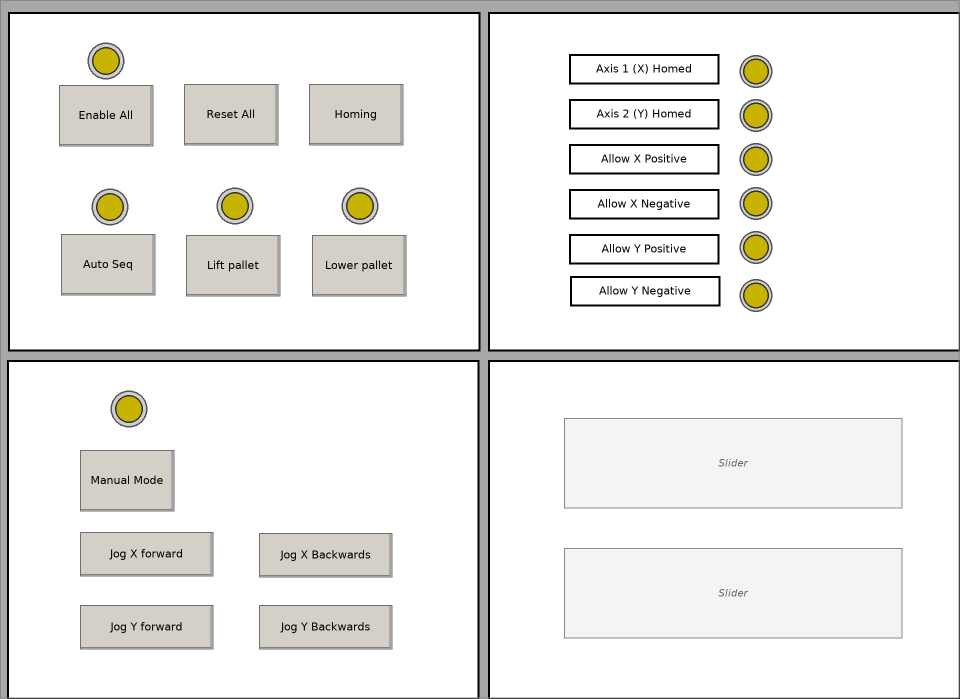
VISUALIZATION Visualization  // 960x699
    Rectangle (8,12 472x339)
    Rectangle (7,360 472x339)
    Rectangle (488,360 472x339)
    Rectangle (488,12 472x339)
    Button (59,85 94x61), "Enable All", colour toggle: GVL_Motion.bEnableAll, pressed state: GVL_Motion.bEnableAll
        OnMouseClick: toggle GVL_Motion.bEnableAll
    Button (184,84 94x61), "Reset All", colour toggle: GVL_Motion.bResetAll
        tap GVL_Motion.bResetAll
    Button (80,450 94x61), "Manual Mode", pressed state: GVL_Motion.bManualModeActive
        OnMouseClick: toggle GVL_Motion.bManualModeActive
    Button (61,234 94x61), "Auto Seq", pressed state: GVL_Motion.bStartAutoseq
        OnMouseClick: execute { GVL_Motion.bStartAutoseq := TRUE; }
    Button (309,84 94x61), "Homing", colour toggle: GVL_Motion.bStartHoming, pressed state: GVL_Motion.bStartHoming
        OnMouseClick: toggle GVL_Motion.bStartHoming
    Lamp1 (85,40 42x42), variable: GVL_Motion.bEnableAll, style: Lamp-Lamp1-Yellow
    Lamp1 (108,388 42x42), variable: GVL_Motion.bManualModeActive, style: Lamp-Lamp1-Yellow
    Button (80,532 133x44), "Jog X forward", pressed state: GVL_Motion.bJogForwardX
        OnMouseDown: toggle GVL_Motion.bJogForwardX
        OnMouseUp: toggle GVL_Motion.bJogForwardX
    Button (259,533 133x44), "Jog X Backwards", pressed state: GVL_Motion.bJogBackwardsX
        OnMouseDown: toggle GVL_Motion.bJogBackwardsX
        OnMouseUp: toggle GVL_Motion.bJogBackwardsX
    Button (80,605 133x44), "Jog Y forward", pressed state: GVL_Motion.bJogForwardY
        OnMouseDown: toggle GVL_Motion.bJogForwardY
        OnMouseUp: toggle GVL_Motion.bJogForwardY
    Button (259,605 133x44), "Jog Y Backwards", pressed state: GVL_Motion.bJogBackwardsY
        OnMouseDown: toggle GVL_Motion.bJogBackwardsY
        OnMouseUp: toggle GVL_Motion.bJogBackwardsY
    Slider (564,418 338x90), variable: GVL_Motion.fVelocityX, scale 0..30
    Slider (564,548 338x90), variable: GVL_Motion.fVelocityY, scale 0..30
    Lamp1 (737,52 38x39), variable: GVL_Motion.bXHomed, style: Lamp-Lamp1-Yellow
    Lamp1 (737,96 38x39), variable: GVL_Motion.bYHomed, style: Lamp-Lamp1-Yellow
    Lamp1 (737,140 38x39), variable: GVL_Motion.bX_Allow_Positive, style: Lamp-Lamp1-Yellow
    Lamp1 (737,184 38x39), variable: GVL_Motion.bX_Allow_Negative, style: Lamp-Lamp1-Yellow
    Lamp1 (737,228 38x39), variable: GVL_Motion.bY_Allow_Positive, style: Lamp-Lamp1-Yellow
    Lamp1 (737,276 38x39), variable: GVL_Motion.bY_Allow_Negative, style: Lamp-Lamp1-Yellow
    Lamp1 (89,186 42x42), variable: GVL_Motion.bSequenceRunning, style: Lamp-Lamp1-Yellow
    Button (186,235 94x61), "Lift pallet", pressed state: GVL_Motion.bRetrievalMode
        OnMouseClick: execute { GVL_Motion.bRetrievalMode := TRUE; }
    Button (312,235 94x61), "Lower pallet", pressed state: NOT GVL_Motion.bRetrievalMode
        OnMouseClick: execute { GVL_Motion.bRetrievalMode := FALSE; }
    Lamp1 (214,185 42x42), variable: GVL_Motion.bRetrievalMode, style: Lamp-Lamp1-Yellow
    Lamp1 (339,185 42x42), variable: NOT GVL_Motion.bRetrievalMode, style: Lamp-Lamp1-Yellow
    Rectangle (570,276 150x30), "Allow Y Negative"
    Rectangle (569,234 150x30), "Allow Y Positive"
    Rectangle (569,189 150x30), "Allow X Negative"
    Rectangle (569,144 150x30), "Allow X Positive"
    Rectangle (569,99 150x30), "Axis 2 (Y) Homed"
    Rectangle (569,54 150x30), "Axis 1 (X) Homed"
END_VISUALIZATION

(* stored: Version 1.1.0.1, ProductVersion 3.1.4024.12
   Visu Visualization: Id {ef786948-4976-4237-8569-45806ceb6a00} *)
